# EPICS substitutions: db/Beckhoff_3XXX/ecmcOptoILD2300_50mm.substitutions
file "ecmcEcSlave.template"
{
  pattern {}
          {}
}

file "ecmcEL3XXX-chX.template"
{
  pattern {CH_ID, LINR,     ESLO,                       EOFF,   EGU,     PREC, LOW, LOLO, HIGH, HIHI, HYST, LLSV,       LSV,        HSV,        HHSV      }
          {1,     "SLOPE",  1e-6,     0,      "V",     0,    0,   0,    0,    0,    0,    "NO_ALARM", "NO_ALARM", "NO_ALARM", "NO_ALARM"}
}
